PROGRAM HMI
VAR
END_VAR

IF MCP_IO.RemoteModeSelected = TRUE (*OR HMI_DB.RemoteModeSelected = TRUE *)THEN 
	GVL.RemoteModeSelected := TRUE;
	ELSE
//ELSIF MCP_IO.RemoteModeSelected = FALSE OR HMI_DB.RemoteModeSelected = FALSE THEN
		GVL.RemoteModeSelected := FALSE;
END_IF

END_PROGRAM

(* stored: Version 1.1.0.1, ProductVersion 3.1.4024.11
   POU HMI: Id {8a79c955-f3ed-4826-b061-613e8797521e}, SpecialFunc None *)
